FUNCTION_BLOCK FB_temppalletpins  IMPLEMENTS temp_ITFPalletPins
VAR_INPUT
END_VAR
VAR_OUTPUT
END_VAR
VAR
	PinsIn :BOOL:= FALSE;
	PinsUit :BOOL := TRUE;
	
END_VAR

{warning 'Add method implementation '}
METHOD Beweegpinsnaarbeneden : bool
END_METHOD

{warning 'Add method implementation '}
METHOD ErinBewegen : bool
END_METHOD

{warning 'Add method implementation '}
METHOD EruitBewegen : bool
END_METHOD

END_FUNCTION_BLOCK

(* stored: Version 1.1.0.1
   POU FB_temppalletpins: Id {24283af4-cc3a-435c-bd24-eb4b86f3a12e}, SpecialFunc None
   Method Beweegpinsnaarbeneden: Id {ceb393c4-911a-42bd-8235-2f86e39d1134}
   Method ErinBewegen: Id {d6ab7a25-1342-4973-aed4-2f65cb559662}
   Method EruitBewegen: Id {51ecdb2a-4d09-46c6-9136-f03523cff8d9} *)
